LIN {X 0,Y 28.793,Z 508.985,A -85,B 0,C 180,E1 -31512.404,E2 -31512.404} C_VEL
LIN {X 0,Y 15.831,Z 510.651,A -85,B 0,C 180,E1 -31527.32,E2 -31527.32} C_VEL
LIN {X 0,Y 7.624,Z 511.226,A -85,B 0,C 180,E1 -31589.933,E2 -31589.933} C_VEL
LIN {X 0,Y 15.806,Z 510.674,A -85,B 0,C 180,E1 -31652.715,E2 -31652.715} C_VEL
LIN {X 0,Y 28.773,Z 509.037,A -85,B 0,C 180,E1 -31667.609,E2 -31667.609} C_VEL
LIN {X 0,Y 42.424,Z 506.254,A -85,B 0,C 180,E1 -31673.586,E2 -31673.586} C_VEL
LIN {X 0,Y 49.343,Z 504.411,A -85,B 0,C 180,E1 -31675.442,E2 -31675.442} C_VEL
LIN {X 0,Y 49.246,Z 504.534,A -85,B 0,C 180,E1 -31677.174,E2 -31677.174} C_VEL
LIN {X 0,Y 35.131,Z 508.261,A -85,B 0,C 180,E1 -31680.288,E2 -31680.288} C_VEL
LIN {X 0,Y 24.298,Z 510.291,A -85,B 0,C 180,E1 -31685.275,E2 -31685.275} C_VEL
LIN {X 0,Y 22.675,Z 512.267,A -85,B 0,C 180,E1 -31686.44,E2 -31686.44} C_VEL
LIN {X 0,Y 22.675,Z 600,A -85,B 0,C 180,E1 -31686.44,E2 -31686.44} C_VEL
LIN {X 0,Y 22.675,Z 600,A -85,B 0,C 180,E1 -31686.44,E2 -31686.44}

QRS_NEXT_CUT()

QRS_NEXT()
QRS_HOME()

END
